(* IEC 61131-3 sources: iolink/src/general (part 3) *)

								// Start Teach Timer
								IF teachTimer <> T#0ms THEN
									instTimer(duration := teachTimer,
									signal := TRUE);
								END_IF;

							ELSIF statRwRecordIOLData.Data[0] = TICMD_TEACH_SP_STOP THEN
								statFBState := FB_STATE_CHECK_RESULT;
								statStatus := STATUS_TEACH_APPLYING; // Busy, Teach process, apply action
							END_IF;

						statMyPermitAbort := TRUE;
						END_IF;
					END_IF;
				END_IF;
				// END_REGION dynamic teach-in

				// REGION check result
				IF statFBState = FB_STATE_CHECK_RESULT THEN
					statMyPermitTeach1 := FALSE;
					statMyPermitTeach2 := FALSE;
					statMyPermitApply := FALSE;
					statMyPermitAbort := FALSE;

					// Read Teach-in state
					instDevice(execute := TRUE,
					readWrite := MODE_READ,
					index := INDEX_TI_RESULT,
					record := statRwRecordIOLData);

					IF instDevice.done THEN
						instDevice(execute := FALSE,
						record := statRwRecordIOLData);

						IF (statRwRecordIOLData.Data[0] AND MASK_TEACH_STATE) = TO_BYTE(TEACH_STATE_BUSY) THEN
							; // Keep trying until teach state of device is not busy
						ELSIF (statRwRecordIOLData.Data[0] AND MASK_TEACH_STATE) = TO_BYTE(TEACH_STATE_SUCCESS) THEN
							statMyPermitTeach1 := FALSE;
							statMyPermitTeach2 := FALSE;
							statMyPermitApply := FALSE;
							statMyPermitAbort := FALSE;

							statFBState := FB_STATE_READ_ALL; // Go to read all
							statIndexRead := INDEX_SSC_PARAM;
							statLenRead := 2;
						ELSIF (statRwRecordIOLData.Data[0] AND MASK_TEACH_STATE) = TO_BYTE(TEACH_STATE_WAIT_FOR_COMMAND) THEN
							statStatus := STATUS_TEACH_WAITING_APPLY;
						ELSIF (statRwRecordIOLData.Data[0] AND MASK_TEACH_STATE) = TO_BYTE(TEACH_STATE_ERROR) THEN
							statStatus := ERR_TEACH_DEVICE;
						END_IF;
					END_IF;
				END_IF;
				// END_REGION check result

				// REGION abort
				// Check for Abort Teach and not permitted Functions
				IF teachRequest AND NOT statTeachRequestOld THEN
					IF teachFunction = TEACH_FUNCTION_1 AND NOT statMyPermitTeach1
						OR teachFunction = TEACH_FUNCTION_2 AND NOT statMyPermitTeach2
						OR teachFunction = TEACH_FUNCTION_APPLY AND NOT statMyPermitApply
						OR teachFunction = TEACH_FUNCTION_ABORT AND NOT statMyPermitAbort
					THEN
						statStatus := ERR_TEACH_NOT_ALLOWED;
					ELSIF teachFunction = TEACH_FUNCTION_ABORT AND statMyPermitAbort THEN
						statFBState := FB_STATE_ABORT_TEACH;
					END_IF;
				END_IF;

				IF statFBState = FB_STATE_ABORT_TEACH THEN
					statStatus := STATUS_TEACH_ABORTING;

					// Abort Teach-in sequence
					statRwRecordIOLData.Data[0] := TICMD_TEACH_CANCEL;
					instDevice(execute := TRUE,
					readWrite := MODE_WRITE,
					index := INDEX_SYS_CMD,
					writeLen := 1,
					record := statRwRecordIOLData);

					IF instDevice.done THEN
						instDevice(execute := FALSE,
						record := statRwRecordIOLData);

						statStatus := STATUS_EXECUTION_FINISHED;
					END_IF;
				END_IF;
				// END_REGION abort

				// Error Handling
				IF instDevice.error THEN
					statStatus := ERR_DEVICE_FB;
					statSubfunctionStatus := instDevice.status;
					statFBErrorState := statFBSubState;
				END_IF;
				// END_REGION teach

			FB_STATE_READ_ALL..FB_STATE_BACKUP:
				// State to read and write Setpoint and Logic

				// REGION read all
				IF statFBState = FB_STATE_READ_ALL THEN // Read "Logic" and "Setpoint"
					statStatus := STATUS_BUSY_READING; // Busy reading data

					instDevice(execute := TRUE,
					readWrite := MODE_READ,
					index := statIndexRead,
					record := statRwRecordIOLData);

					IF instDevice.done THEN
						instDevice(execute := FALSE,
						record := statRwRecordIOLData);

						IF statIndexRead >= INDEX_SSC_CONFIG THEN
							logicOut := TO_BOOL(statRwRecordIOLData.Data[0] AND BYTE#2#00000001);

							IF backupEnable AND functionCmd = FUNC_TEACH THEN
								statFBState := FB_STATE_BACKUP;
							ELSE
								statStatus := STATUS_EXECUTION_FINISHED;
							END_IF;

						ELSE
							tempSetpointOut1.%B0 := statRwRecordIOLData.Data[1];
							tempSetpointOut1.%B1 := statRwRecordIOLData.Data[0];
							setpointOut1 := TO_INT(tempSetpointOut1);

							tempSetpointOut2.%B0 := statRwRecordIOLData.Data[1];
							tempSetpointOut2.%B1 := statRwRecordIOLData.Data[0];
							setpointOut2 := TO_INT(tempSetpointOut2);

							// Read "Logic" after reading "Setpoint"
							statIndexRead := statIndexRead + (1);
							statLenRead := 1;
						END_IF;
					END_IF;
				END_IF;
				// END_REGION read all

				// REGION write config
				IF statFBState = FB_STATE_WRITE_CONF THEN
					statStatus := STATUS_BUSY_WRITING; // Busy writing data
					statRwRecordIOLData.Data[0] := TO_BYTE(logicIn);

					instDevice(execute := true,
						readWrite := MODE_WRITE,
						index := INDEX_SSC_CONFIG,
						writeLen := 1,
						record := statRwRecordIOLData);

					IF instDevice.done THEN
						//Write input to output if writing was successful
						logicOut := logicIn;

						IF backupEnable THEN
							statFBState := FB_STATE_BACKUP;
							instDevice(execute := FALSE,
							record := statRwRecordIOLData);
						ELSE
							statStatus := STATUS_EXECUTION_FINISHED;
						END_IF;
					END_IF;
				END_IF;
				// END_REGION write config

				// REGION write param
				IF statFBState = FB_STATE_WRITE_PARAM THEN
					statStatus := STATUS_BUSY_WRITING;

					tempSetpointIn1 := TO_WORD(setpointIn1);
					statRwRecordIOLData.Data[1] := tempSetpointIn1.%B0;
					statRwRecordIOLData.Data[0] := tempSetpointIn1.%B1;

					tempSetpointIn2 := TO_WORD(setpointIn2);
					statRwRecordIOLData.Data[1] := tempSetpointIn2.%B0;
					statRwRecordIOLData.Data[0] := tempSetpointIn2.%B1;

					instDevice(execute := TRUE,
					readWrite := MODE_WRITE,
					index := INDEX_SSC_PARAM,
					writeLen := 2,
					record := statRwRecordIOLData);

					IF instDevice.done THEN
						//Write input to output if writing was successful
						setpointOut1 := setpointIn1;
						setpointOut2 := setpointIn2;
						IF backupEnable THEN
							statFBState := FB_STATE_BACKUP;
							instDevice(execute := FALSE,
							record := statRwRecordIOLData);
						ELSE
							statStatus := STATUS_EXECUTION_FINISHED;
						END_IF;
					END_IF;
				END_IF;
				// END_REGION write param

				// REGION param download store
				IF statFBState = FB_STATE_BACKUP THEN
					statStatus := STATUS_BUSY_BACKUP; // Busy backup
					statRwRecordIOLData.Data[0] := BYTE#16#05;

					instDevice(execute := TRUE,
					readWrite := MODE_WRITE,
					index := INDEX_SYS_CMD,
					writeLen := 1,
					record := statRwRecordIOLData);

					IF instDevice.done THEN
						statStatus := STATUS_EXECUTION_FINISHED;
					END_IF;
				END_IF;
				// END_REGION param download store

				// Error handling
				IF instDevice.error THEN
					statStatus := ERR_DEVICE_FB;
					statSubfunctionStatus := instDevice.status;
					statFBErrorState := statFBState;
				END_IF;
				// END_REGION param exchange
		END_CASE;
		// END_REGION STATE_MACHINE

		// REGION OUTPUTS
		// Write outputs
		IF (statStatus = STATUS_EXECUTION_FINISHED) AND (statDone = FALSE) THEN // Execution finished without errors
			// REGION execution finished
			statDone := TRUE;
			statBusy := FALSE;
			statError := FALSE;

			statMyPermitTeach1 := FALSE;
			statMyPermitTeach2 := FALSE;
			statMyPermitApply := FALSE;
			statMyPermitAbort := FALSE;

			// execution aborted --> set state no processing
			statFBState := FB_STATE_NO_PROCESSING;
			statFBState := 0;
			statFBSubState := 0;
			// END_REGION execution finished

		ELSIF (statStatus.%X15 = TRUE) AND (statError = FALSE) THEN // Error occurred (#statStatus is 16#8000 to 16#FFFF)
			// REGION error occured
			statDone := FALSE;
			statBusy := FALSE;
			statError := TRUE;

			statMyPermitTeach1 := FALSE;
			statMyPermitTeach2 := FALSE;
			statMyPermitApply := FALSE;
			statMyPermitAbort := FALSE;

			// Write diagnostics
			diagnostics.status := statStatus;
			diagnostics.subfunctionStatus := statSubfunctionStatus;
			diagnostics.stateNumber := statFBErrorState;

			// Reset instance for next job
			instDevice(execute := FALSE,
			record := statRwRecordIOLData);

			// execution aborted --> set state no processing
			statFBState := FB_STATE_NO_PROCESSING;
			statFBState := 0;
			statFBSubState := 0;
			// END_REGION error occured

		ELSIF (tempExecute = FALSE) AND ((statDone = TRUE) OR (statError = TRUE)) THEN // Reset outputs
			// REGION execute reset
			statDone := FALSE;
			statBusy := FALSE;
			statError := FALSE;
			statStatus := STATUS_NO_CALL;

			// Reset instance for next job
			instDevice(execute := FALSE,
			record := statRwRecordIOLData);

			// END_REGION execute reset
		END_IF;

		// REGION Write static values to outputs
		done := statDone;
		busy := statBusy;
		error := statError;
		status := statStatus;

		// Write internal used variables to outputs
		permitTeach1 := statMyPermitTeach1;
		permitTeach2 := statMyPermitTeach2;
		permitApply := statMyPermitApply;
		permitAbort := statMyPermitAbort;

		// Needed to detect rising edge at inputs
		statTeachRequestOld := teachRequest;

		// END_REGION Write static values to outputs
		// END_REGION OUTPUTS
	END_FUNCTION_BLOCK

	TYPE
		statIdentObjectInfoType : STRUCT   // Contains information about the elements of output IdentificationObjects
			index : Int := 0;   // Index of parameter
			len : Int := 12;   // Length of parameter
			optional : Bool := false;   // Parameter is optional
		END_STRUCT;
	END_TYPE

END_NAMESPACE
